ABB RobotStudio station: simulation of path.rsstn

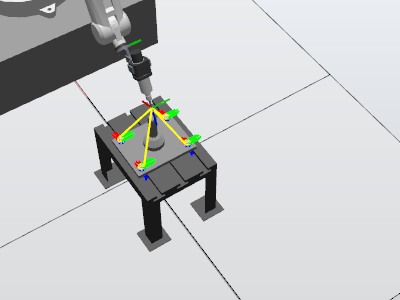
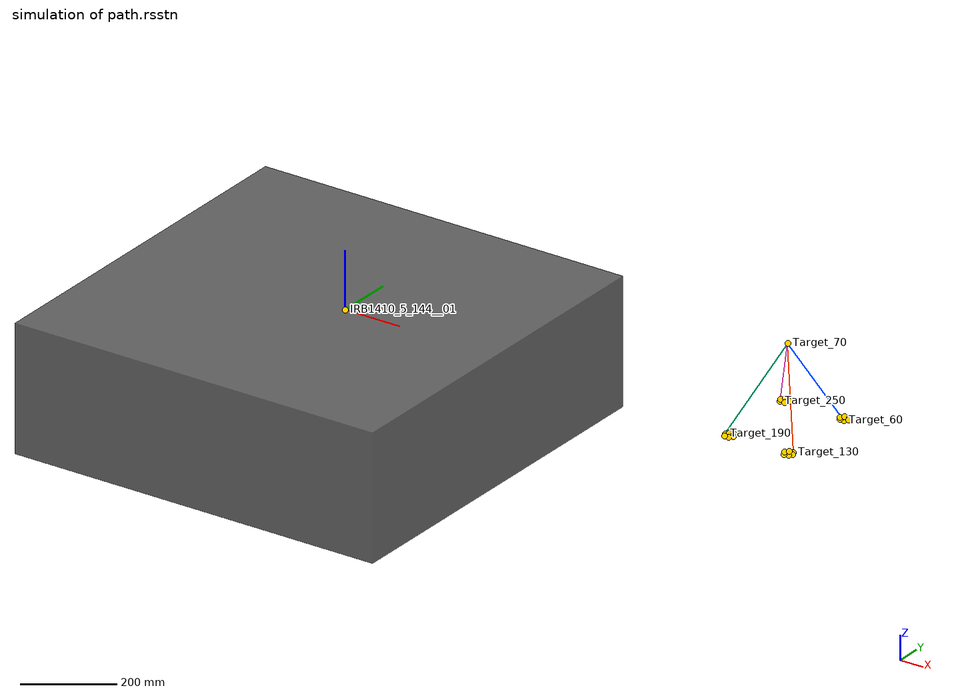
[picture v1: parts stored in the station drawn from their meshes, with robot base, taught points and paths (robot models come from the ABB library and are not in the file)]
Station simulation of path (saved by RobotStudio 22.3.10141.1)
Controller Controller13, task T_ROB1: task frame (RAPID world) sits at (0, 0, 292.3) mm in the station
Controller Controller13
  mechanical unit ROB_1: IRB1410_5_144__01, 6 joints, base frame (0, 0, 0) mm
Layout (positions relative to the parent item):
  - IRB1410_5_144__01 [mechanism, from Robots\IRB1410_5_144_G_01.rslib] at (0, 0, 292.3) mm; joint values [0.0023, 0.4782, 1.1051, 0.0036, -0.5815, -0.0019] (rad or m)
  - MyTool [mechanism, from Training Objects\myTool.rslib] at (930.24, 1.94, 668.02) mm, rotated rx -180 ry 60 rz -180 deg
  - Part_1 [part] at (-513.88, -453.3, 0) mm, size 900 x 900 x 300 mm
  - table_and_fixture_140 [part, from Training Objects\propeller_table.rslib] at (886.99, -175, 0) mm
Attachment: MyTool is attached to IRB1410_5_144__01 / Link6
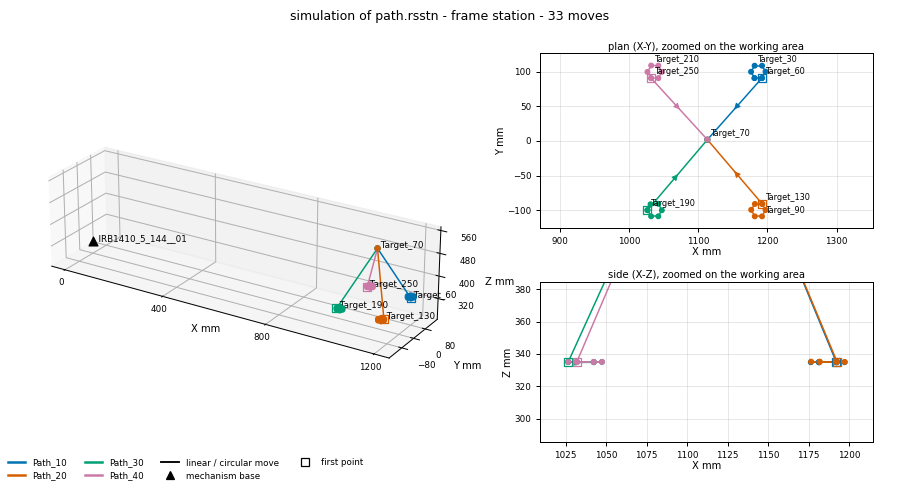
[picture p0: tool path of simulation of path.rsstn in frame station, 33 of 33 moves have a stored position in this frame; points joined in program order, loops and branches not executed]
Targets, tools, work objects and paths stored in the station, written as RAPID:
! task T_ROB1
MODULE CalibData
  PERS tooldata MyTool:=[TRUE,[[31.792631019,0,229.638935148],[0.945518576,0,0.325568154,0]],[1,[0,0,1],[1,0,0,0],0,0,0]];
ENDMODULE

! task T_ROB1
MODULE Module1
  CONST robtarget Target_10:=[[1181.347997327,90.953695559,42.596489658],[0.190807769,0.000000024,0.981627422,-0.000000027],[0,0,-1,0],[9E+09,9E+09,9E+09,9E+09,9E+09,9E+09]];
  CONST robtarget Target_20:=[[1176.347974723,100.112008436,42.596494387],[0.190807429,0.000000028,0.981627488,-0.000000024],[0,0,-1,0],[9E+09,9E+09,9E+09,9E+09,9E+09,9E+09]];
  CONST robtarget Target_30:=[[1181.478000962,108.867998541,42.596458551],[0.190807138,0.000000021,0.981627544,-0.000000026],[0,0,-1,0],[9E+09,9E+09,9E+09,9E+09,9E+09,9E+09]];
  CONST robtarget Target_40:=[[1192.255041516,108.868000766,42.596449078],[0.190806944,0.000000014,0.981627582,-0.000000027],[0,0,-1,0],[9E+09,9E+09,9E+09,9E+09,9E+09,9E+09]];
  CONST robtarget Target_50:=[[1197.235927375,100.298297956,42.596557682],[0.190806761,0.000000011,0.981627618,-0.000000022],[0,0,-1,0],[9E+09,9E+09,9E+09,9E+09,9E+09,9E+09]];
  CONST robtarget Target_60:=[[1192.137917793,91.017993798,42.596479663],[0.190806524,0.000000006,0.981627664,-0.000000027],[0,0,-1,0],[9E+09,9E+09,9E+09,9E+09,9E+09,9E+09]];
  CONST robtarget Target_70:=[[1113.219942379,1.941895077,233.37111167],[0.190806219,0.000000016,0.981627723,-0.000000022],[0,0,-1,0],[9E+09,9E+09,9E+09,9E+09,9E+09,9E+09]];
  CONST robtarget Target_80:=[[1197.314912189,-99.827185107,42.769556202],[0.190805109,0.000000012,0.981627939,-0.00000003],[-1,-1,0,0],[9E+09,9E+09,9E+09,9E+09,9E+09,9E+09]];
  CONST robtarget Target_90:=[[1192.224951852,-108.972688573,42.769554783],[0.190805041,0.000000012,0.981627952,-0.000000032],[-1,-1,0,0],[9E+09,9E+09,9E+09,9E+09,9E+09,9E+09]];
  CONST robtarget Target_100:=[[1181.738961886,-108.972693705,42.769572184],[0.190804965,0.000000015,0.981627967,-0.00000003],[-1,-1,0,0],[9E+09,9E+09,9E+09,9E+09,9E+09,9E+09]];
  CONST robtarget Target_110:=[[1176.519930655,-99.52934193,42.946808071],[0.190804489,0.000000028,0.981628059,-0.000000034],[-1,-1,0,0],[9E+09,9E+09,9E+09,9E+09,9E+09,9E+09]];
  CONST robtarget Target_120:=[[1181.893007517,-91.028141487,42.946808503],[0.190804254,0.000000031,0.981628105,-0.000000035],[-1,-1,0,0],[9E+09,9E+09,9E+09,9E+09,9E+09,9E+09]];
  CONST robtarget Target_130:=[[1192.509069001,-91.028134918,42.94680837],[0.190804245,0.000000027,0.981628107,-0.000000035],[-1,-1,0,0],[9E+09,9E+09,9E+09,9E+09,9E+09,9E+09]];
  CONST robtarget Target_140:=[[1030.972018039,-91.499642652,42.442201301],[0.190802259,-0.000000022,0.981628493,-0.000000039],[-1,-1,0,0],[9E+09,9E+09,9E+09,9E+09,9E+09,9E+09]];
  CONST robtarget Target_150:=[[1042.242982911,-90.823635311,42.552283951],[0.190801317,-0.00000002,0.981628676,-0.000000025],[-1,-1,0,0],[9E+09,9E+09,9E+09,9E+09,9E+09,9E+09]];
  CONST robtarget Target_160:=[[1047.323922387,-100.13468964,42.799108785],[0.190801032,-0.000000021,0.981628731,-0.000000032],[-1,-1,0,0],[9E+09,9E+09,9E+09,9E+09,9E+09,9E+09]];
  CONST robtarget Target_170:=[[1042.263932198,-108.878391796,42.799097378],[0.190800715,-0.000000016,0.981628793,-0.00000003],[-1,-1,0,0],[9E+09,9E+09,9E+09,9E+09,9E+09,9E+09]];
  CONST robtarget Target_180:=[[1031.834911054,-108.878387805,42.799111443],[0.190800611,-0.000000017,0.981628813,-0.00000003],[-1,-1,0,0],[9E+09,9E+09,9E+09,9E+09,9E+09,9E+09]];
  CONST robtarget Target_190:=[[1026.530031981,-100.040699048,42.799117067],[0.190800365,-0.000000014,0.981628861,-0.000000028],[-1,-1,0,0],[9E+09,9E+09,9E+09,9E+09,9E+09,9E+09]];
  CONST robtarget Target_200:=[[1026.530043615,99.910160372,42.799219207],[0.190800375,-0.000000025,0.981628859,-0.000000041],[0,0,-1,0],[9E+09,9E+09,9E+09,9E+09,9E+09,9E+09]];
  CONST robtarget Target_210:=[[1031.901960904,109.137895077,42.799275195],[0.190800143,-0.000000037,0.981628904,-0.000000039],[0,0,-1,0],[9E+09,9E+09,9E+09,9E+09,9E+09,9E+09]];
  CONST robtarget Target_220:=[[1042.330038494,109.004290642,42.799320111],[0.190799736,-0.000000026,0.981628983,-0.000000036],[0,0,-1,0],[9E+09,9E+09,9E+09,9E+09,9E+09,9E+09]];
  CONST robtarget Target_230:=[[1047.381982246,99.986447475,42.799316628],[0.190799337,-0.00000003,0.981629061,-0.000000036],[0,0,-1,0],[9E+09,9E+09,9E+09,9E+09,9E+09,9E+09]];
  CONST robtarget Target_240:=[[1042.274038265,90.887192568,42.729635382],[0.190798358,-0.000000055,0.981629251,-0.00000003],[0,0,-1,0],[9E+09,9E+09,9E+09,9E+09,9E+09,9E+09]];
  CONST robtarget Target_250:=[[1031.808011159,90.887183128,42.72964561],[0.190798123,-0.000000056,0.981629297,-0.00000003],[0,0,-1,0],[9E+09,9E+09,9E+09,9E+09,9E+09,9E+09]];
  CONST robtarget Target_260:=[[1192.137894866,91.017983448,42.59650643],[0.190806524,0.000000018,0.981627664,-0.000000018],[0,0,-1,0],[9E+09,9E+09,9E+09,9E+09,9E+09,9E+09]];
  PROC Path_10()
    MoveL Target_60,v1000,fine,MyTool\WObj:=wobj0;
    MoveL Target_10,v1000,fine,MyTool\WObj:=wobj0;
    MoveL Target_10,v1000,fine,MyTool\WObj:=wobj0;
    MoveL Target_20,v1000,fine,MyTool\WObj:=wobj0;
    MoveL Target_30,v1000,fine,MyTool\WObj:=wobj0;
    MoveL Target_40,v1000,fine,MyTool\WObj:=wobj0;
    MoveL Target_50,v1000,fine,MyTool\WObj:=wobj0;
    MoveL Target_60,v1000,fine,MyTool\WObj:=wobj0;
    MoveL Target_70,v1000,z100,MyTool\WObj:=wobj0;
  ENDPROC
  PROC Path_20()
    MoveL Target_130,v1000,fine,MyTool\WObj:=wobj0;
    MoveL Target_80,v1000,fine,MyTool\WObj:=wobj0;
    MoveL Target_90,v1000,fine,MyTool\WObj:=wobj0;
    MoveL Target_100,v1000,fine,MyTool\WObj:=wobj0;
    MoveL Target_110,v1000,fine,MyTool\WObj:=wobj0;
    MoveL Target_120,v1000,fine,MyTool\WObj:=wobj0;
    MoveL Target_130,v1000,fine,MyTool\WObj:=wobj0;
    MoveL Target_70,v1000,fine,MyTool\WObj:=wobj0;
  ENDPROC
  PROC Path_30()
    MoveL Target_190,v1000,fine,MyTool\WObj:=wobj0;
    MoveL Target_140,v1000,fine,MyTool\WObj:=wobj0;
    MoveL Target_150,v1000,fine,MyTool\WObj:=wobj0;
    MoveL Target_160,v1000,fine,MyTool\WObj:=wobj0;
    MoveL Target_170,v1000,fine,MyTool\WObj:=wobj0;
    MoveL Target_180,v1000,fine,MyTool\WObj:=wobj0;
    MoveL Target_190,v1000,fine,MyTool\WObj:=wobj0;
    MoveL Target_70,v1000,fine,MyTool\WObj:=wobj0;
  ENDPROC
  PROC Path_40()
    MoveL Target_250,v1000,fine,MyTool\WObj:=wobj0;
    MoveL Target_200,v1000,fine,MyTool\WObj:=wobj0;
    MoveL Target_210,v1000,fine,MyTool\WObj:=wobj0;
    MoveL Target_220,v1000,fine,MyTool\WObj:=wobj0;
    MoveL Target_230,v1000,fine,MyTool\WObj:=wobj0;
    MoveL Target_240,v1000,fine,MyTool\WObj:=wobj0;
    MoveL Target_250,v1000,fine,MyTool\WObj:=wobj0;
    MoveL Target_70,v1000,fine,MyTool\WObj:=wobj0;
  ENDPROC
  PROC Path_50()
    Path_10;
    Path_20;
    Path_30;
    Path_40;
  ENDPROC
ENDMODULE

